// TwinCAT 3 PLC project ElevatorController
// ProgramVersion: 3.1.4023.0
// libraries:
//   Tc2_Standard, * (Beckhoff Automation GmbH)
//   Tc2_System, * (Beckhoff Automation GmbH)
//   Tc3_Module, * (Beckhoff Automation GmbH)
// project tree:
//   DUT/ E_States.TcDUT (not stored), ST_LevelSensors.TcDUT
//   / GlobalTextList.TcGTLO, Visualization Manager.TcVMO (not stored)
//   POU/ FB_Motor.TcPOU (not stored), MAIN.TcPOU
//   Tasks/ PlcTask.TcTTO (not stored), VISU_TASK.TcTTO
//   VISU/ CallButtons.TcVIS, Floor.TcVIS, Screen3.TcVIS, Screen2.TcVIS, Screen1.TcVIS, Visualization.TcVIS
// real-time tasks:
//   TASK PlcTask: cycle T#20ms, priority 20, ADS port 350
//   TASK HIL Task: cycle T#10ms, priority 21, ADS port 351
//   TASK VISU_TASK: cycle T#50000us, priority 30, ADS port 352
// I/O:
//   DEVICE Device 1 (EtherCAT) (disabled), AmsNetId 169.254.141.45.2.1
//     Term 1 (EK1100) [EK1100 EtherCAT Coupler (2A E-Bus)]
//       Term 2 (EL1809) [EL1809 16Ch. Dig. Input 24V, 3ms]
//       Term 3 (EL2004) [EL2004 4Ch. Dig. Output 24V, 0.5A]
// variable links:
//   ElevatorController/ElevatorController Instance <-> HIL Simulation/HIL Simulation Instance
//     PlcTask Inputs/MAIN.LS_Floor[1]/High <-> PlcTask Outputs/MAIN.LS_Floor[1]/High
//     PlcTask Inputs/MAIN.LS_Floor[2]/High <-> PlcTask Outputs/MAIN.LS_Floor[2]/High
//     PlcTask Inputs/MAIN.LS_Floor[3]/High <-> PlcTask Outputs/MAIN.LS_Floor[3]/High
//     PlcTask Inputs/MAIN.LS_Floor[1]/Low <-> PlcTask Outputs/MAIN.LS_Floor[1]/Low
//     PlcTask Inputs/MAIN.LS_Floor[2]/Low <-> PlcTask Outputs/MAIN.LS_Floor[2]/Low
//     PlcTask Inputs/MAIN.LS_Floor[3]/Low <-> PlcTask Outputs/MAIN.LS_Floor[3]/Low
//     PlcTask Inputs/MAIN.LS_Floor[1]/Mid <-> PlcTask Outputs/MAIN.LS_Floor[1]/Mid
//     PlcTask Inputs/MAIN.LS_Floor[2]/Mid <-> PlcTask Outputs/MAIN.LS_Floor[2]/Mid
//     PlcTask Inputs/MAIN.LS_Floor[3]/Mid <-> PlcTask Outputs/MAIN.LS_Floor[3]/Mid
//     PlcTask Outputs/MAIN.CurrentFloor <-> PlcTask Inputs/MAIN.CurrentFloor
//     PlcTask Outputs/MAIN.Elevator.Brake <-> PlcTask Inputs/MAIN.Motor/Brake
//     PlcTask Outputs/MAIN.Elevator.Down <-> PlcTask Inputs/MAIN.Motor/Down
//     PlcTask Outputs/MAIN.Elevator.Slow <-> PlcTask Inputs/MAIN.Motor/Slow
//     PlcTask Outputs/MAIN.Elevator.Up <-> PlcTask Inputs/MAIN.Motor/Up
//     PlcTask Outputs/MAIN.RequestedFloor <-> PlcTask Inputs/MAIN.RequestedFloor

CONFIGURATION ElevatorController
    RESOURCE PLC ON TwinCAT3
        TASK VISU_TASK(INTERVAL := T#50000us, PRIORITY := 30);
        PROGRAM VisuElems_Visu_Prg WITH VISU_TASK : VisuElems.Visu_Prg;
    END_RESOURCE
END_CONFIGURATION

// ---- DUT/ST_LevelSensors.TcDUT
TYPE ST_LevelSensors :
STRUCT
	Low,
	Mid,
	High :BOOL;
END_STRUCT
END_TYPE

// ---- POU/MAIN.TcPOU
PROGRAM MAIN
VAR
	LS_Floor AT %I*:ARRAY[1..3]	OF	ST_LevelSensors;
	BT_FloorCall :ARRAY[1..3]	OF	BOOL;
	Elevator:FB_Motor;
	STATE: E_States;
	RequestedFloor AT%Q*: INT;
	CurrentFloor AT%Q*:INT;
	i: INT;
	PulseTrigger:ARRAY[1..3]OF	R_Trig;
	LatchTime: ULINT;
	ElapsedTime: LTIME;
END_VAR


CASE STATE	OF	
	E_States.Call:;
		//action logic
		FOR	i:=1 TO 3	DO
			IF	BT_FloorCall[i]	THEN
				RequestedFloor:=i;
				EXIT;
			END_IF
		END_FOR
		//transitions
		IF	RequestedFloor>CurrentFloor	THEN
			STATE:=E_States.MoveUp;
		ELSIF	RequestedFloor<CurrentFloor	THEN
			STATE:=E_States.MoveDown;
		END_IF
		
		//initialise pulse timer
		FOR	i:=1	TO	3	DO
			PulseTrigger[i](CLK:=FALSE);
		END_FOR
		
	E_States.MoveUp:
		Elevator.MoveUp();
		FOR	i:=1	TO	3	DO
			PulseTrigger[i](CLK:=LS_Floor[i].Low);
			IF	PulseTrigger[i].Q	THEN
				STATE:=E_States.IncrementFloor;
			END_IF
		END_FOR
		IF	RequestedFloor=CurrentFloor	THEN	
			state:=E_States.SlowDown;
		END_IF
		
	E_States.MoveDown:
		Elevator.MoveDown();
		FOR	i:=1	TO	3	DO
			PulseTrigger[i](CLK:=LS_Floor[i].High);
			IF	PulseTrigger[i].Q	THEN
				STATE:=E_States.DecrementFloor;
			END_IF
		END_FOR
		IF	RequestedFloor=CurrentFloor	THEN	
			state:=E_States.SlowDown;
		END_IF
		
	E_States.IncrementFloor:
		CurrentFloor:=CurrentFloor+1;
		STATE:=E_States.MoveUp;
	E_States.DecrementFloor:
		CurrentFloor:=CurrentFloor-1;
		STATE:=E_States.MoveDown;
	E_States.SlowDown:
		Elevator.SlowDown();
		FOR	i:=1	TO	3	DO
			IF	LS_Floor[i].Mid	THEN
				STATE:=E_States.Stop;
			END_IF
		END_FOR
	E_States.Stop:
		//ElapsedTime:=ULINT_TO_LTIME(F_GetSystemTime()-LatchTime);
		Elevator.Stop();
		state:=E_States.Call;
END_CASE

END_PROGRAM

// ---- GlobalTextList.TcGTLO
TEXTLIST GlobalTextList
  299 = 'Call L1'
  388 = 'Call L2'
  731 = 'Call L3'
  735 = 'Call Level 1'
  22 = 'Call Level 2'
  772 = 'Call Level 3'
  369 = 'Floor 1 status'
  71 = 'Floor 2 status'
  458 = 'Floor 3 status'
  570 = 'High'
  962 = 'Low'
  607 = 'Mid'
END_TEXTLIST

// ---- VISU/CallButtons.TcVIS
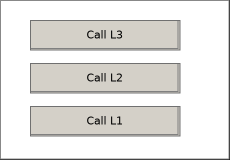
VISUALIZATION CallButtons  // 230x160
VAR_IN_OUT
	L1Call,
	L2Call,
	L3Call:BOOL;
END_VAR
    Rectangle (0,0 230x160)
    Button (30,20 150x30), "Call L3"
        tap L3Call
    Button (30,63 150x30), "Call L2"
        tap L2Call
    Button (30,106 150x30), "Call L1"
        tap L1Call
END_VISUALIZATION

// ---- VISU/Floor.TcVIS
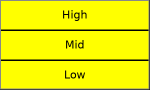
VISUALIZATION Floor  // 150x90
VAR_INPUT
	LS_Floor :ST_LevelSensors;
END_VAR
    Rectangle (0,60 150x30), "Low", colour toggle: LS_Floor.Low
    Rectangle (0,30 150x30), "Mid", colour toggle: LS_Floor.Mid
    Rectangle (0,0 150x30), "High", colour toggle: LS_Floor.High
END_VISUALIZATION

// ---- VISU/Screen3.TcVIS
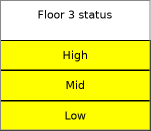
VISUALIZATION Screen3  // 151x131
    Frame (0,40 151x91)
        shows Floor(LS_Floor := MAIN.LS_Floor[3])
        OnMouseClick: change screen: Previous 
    Label (0,0 150x30), "Floor 3 status"
END_VISUALIZATION

// ---- VISU/Screen2.TcVIS
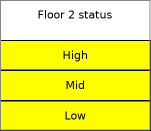
VISUALIZATION Screen2  // 151x131
    Frame (0,40 151x91)
        shows Floor(LS_Floor := MAIN.LS_Floor[2])
        OnMouseClick: change screen: Previous 
    Label (0,0 150x30), "Floor 2 status"
END_VISUALIZATION

// ---- VISU/Screen1.TcVIS
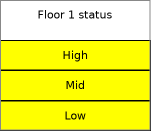
VISUALIZATION Screen1  // 151x131
    Frame (0,40 151x91)
        shows Floor(LS_Floor := MAIN.LS_Floor[1])
        OnMouseClick: change screen: Previous 
    Label (0,0 150x30), "Floor 1 status"
END_VISUALIZATION

// ---- VISU/Visualization.TcVIS
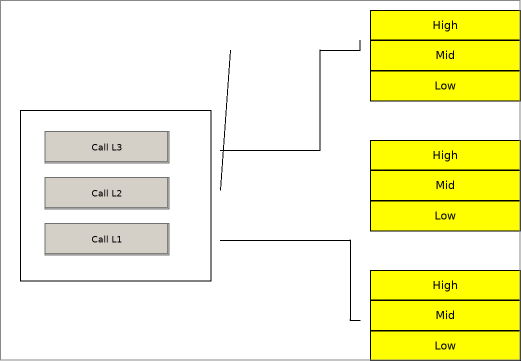
VISUALIZATION Visualization  // 521x361
    Frame (20,110 191x171)
        shows CallButtons(L1Call := MAIN.BT_FloorCall[1], L2Call := MAIN.BT_FloorCall[2], L3Call := MAIN.BT_FloorCall[3])
    Frame (370,10 151x91)
        shows Floor(LS_Floor := MAIN.LS_Floor[3])
        OnMouseClick: change screen: Screen3
    Frame (370,140 151x91)
        shows Floor(LS_Floor := MAIN.LS_Floor[2])
        OnMouseClick: change screen: Screen2
    Frame (370,270 151x91)
        shows Floor(LS_Floor := MAIN.LS_Floor[1])
        OnMouseClick: change screen: Screen1
    Polyline (220,150) (320,150) (320,50) (360,50) (360,40)
    Line (230,50) (220,190)
    Polyline (220,240) (350,240) (350,320) (360,320)
END_VISUALIZATION
